// TIA Portal V18 export
DATA_BLOCK "ProcessData_1"   // DB2300
{ S7_Optimized_Access := 'FALSE' }
VERSION : 0.1
// stored: AutoNumber false, DBAccessibleFromOPCUA true, DBAccessibleFromWebserver true, IsOnlyStoredInLoadMemory false, IsWriteProtectedInAS false
   VAR RETAIN
      AlwaysZero : Byte := 16#00;
      "OP40.2" : Struct
         Kistler_Continue_Interlock : Bool := FALSE;
         Kistler_Interlock : Bool := FALSE;
         KistlerPress_autoInterlock : Bool := FALSE;
         KistlerPress_1Flag : Bool := FALSE;
         KistlerPress_2Flag : Bool := FALSE;
         KistlerPress_1Flag_Reset : Bool := FALSE;
         KistlerPress_2Flag_Reset : Bool := FALSE;
         Spare_7 : Bool := FALSE;
         Spare_8 : Bool := FALSE;
         Spare_9 : Bool := FALSE;
         Spare_10 : Bool := FALSE;
         Spare_11 : Bool := FALSE;
         Spare_12 : Bool := FALSE;
         Spare_13 : Bool := FALSE;
         Spare_14 : Bool := FALSE;
         Spare_15 : Bool := FALSE;
      END_STRUCT;
      "OP40.3" : Struct
         Kistler_Continue_Interlock : Bool := FALSE;
         Kistler_Interlock : Bool := FALSE;
         KistlerPress_autoInterlock : Bool := FALSE;
         KistlerPress_1Flag : Bool := FALSE;
         KistlerPress_2Flag : Bool := FALSE;
         KistlerPress_1Flag_Reset : Bool := FALSE;
         KistlerPress_2Flag_Reset : Bool := FALSE;
         Spare_7 : Bool := FALSE;
         Spare_8 : Bool := FALSE;
         Spare_9 : Bool := FALSE;
         Spare_10 : Bool := FALSE;
         Spare_11 : Bool := FALSE;
         Spare_12 : Bool := FALSE;
         Spare_13 : Bool := FALSE;
         Spare_14 : Bool := FALSE;
         Spare_15 : Bool := FALSE;
      END_STRUCT;
      "HMI_OP40.2" { S7_SetPoint := 'True'} : "OP40_Data";
      "HMI_OP40.3" { S7_SetPoint := 'True'} : "OP40_Data";
      PressInterlock_1 { S7_SetPoint := 'True'} : Array[0..15] of Bool;
      PressInterlock_2 : Array[0..15] of Bool;
      Calibartion_1 : Bool;
      Calibartion_2 : Bool;
   END_VAR
BEGIN
   "HMI_OP40.2".AssemblyResult := 16#00;
   "HMI_OP40.2".SN := '';
   "HMI_OP40.2".ProcessData.AssemblyResult1 := 16#00;
   "HMI_OP40.2".ProcessData.AssemblyResult2 := 16#00;
   "HMI_OP40.2".ProcessData.StartForce1 := 0.0;
   "HMI_OP40.2".ProcessData.StartLVDT1 := 0.0;
   "HMI_OP40.2".ProcessData.ProcessForce1 := 0.0;
   "HMI_OP40.2".ProcessData.ProcessLVDT1 := 0.0;
   "HMI_OP40.2".ProcessData.EndForce1 := 0.0;
   "HMI_OP40.2".ProcessData.EndLVDT1 := 0.0;
   "HMI_OP40.2".ProcessData.StartForce2 := 0.0;
   "HMI_OP40.2".ProcessData.StartLVDT2 := 0.0;
   "HMI_OP40.2".ProcessData.ProcessForce2 := 0.0;
   "HMI_OP40.2".ProcessData.ProcessLVDT2 := 0.0;
   "HMI_OP40.2".ProcessData.EndForce2 := 0.0;
   "HMI_OP40.2".ProcessData.EndLVDT2 := 0.0;
   "HMI_OP40.3".AssemblyResult := 16#00;
   "HMI_OP40.3".SN := '';
   "HMI_OP40.3".ProcessData.AssemblyResult1 := 16#00;
   "HMI_OP40.3".ProcessData.AssemblyResult2 := 16#00;
   "HMI_OP40.3".ProcessData.StartForce1 := 0.0;
   "HMI_OP40.3".ProcessData.StartLVDT1 := 0.0;
   "HMI_OP40.3".ProcessData.ProcessForce1 := 0.0;
   "HMI_OP40.3".ProcessData.ProcessLVDT1 := 0.0;
   "HMI_OP40.3".ProcessData.EndForce1 := 0.0;
   "HMI_OP40.3".ProcessData.EndLVDT1 := 0.0;
   "HMI_OP40.3".ProcessData.StartForce2 := 0.0;
   "HMI_OP40.3".ProcessData.StartLVDT2 := 0.0;
   "HMI_OP40.3".ProcessData.ProcessForce2 := 0.0;
   "HMI_OP40.3".ProcessData.ProcessLVDT2 := 0.0;
   "HMI_OP40.3".ProcessData.EndForce2 := 0.0;
   "HMI_OP40.3".ProcessData.EndLVDT2 := 0.0;
END_DATA_BLOCK
